PROGRAM MAIN
VAR
END_VAR

END_PROGRAM

(* stored: Version 1.1.0.1
   POU MAIN: Id {ce72eb47-a814-467a-b555-3bad272166b0} *)
